// TIA Portal V21 export
FUNCTION "GestGruppoValvoleFestoVTEM" : Void   // FC68, LAD
{ S7_Optimized_Access := 'TRUE' }
// Ogni gruppo valvole festo può portare 8 valvole.
// Ognuno di qusti slot utilizza 3. word in lettura e 3 word in scrittura.
// 
// Se non vengono utilizzate 8 valvole è possibile sfruttura i moduli liberi per leggere dei dati dalle valvole. é anche possibile la lettura e scrittura ciclica delle informazioni.
// stored: SetENOAutomatically false
   VAR_INPUT
      HW_SUBMODULE : HW_SUBMODULE;
      SLOT01_K_Tipo : Int;
      SLOT01_K_UtenzaAttuatore : Int;   // Dichiarare la costante ad esempio k_valvolafestovftem oppure k_analogica da assegnare allo slot
      SLOT02_K_Tipo : Int;   // Dichiarare l'utilizzo dello slot, se deve essere utilizzato per leggere le informazioni dichiarare TipoAnalogica altrimenti valvola
      SLOT02_K_UtenzaAttuatore : Int;   // Dichiarare la costante ad esempio k_valvolafestovftem oppure k_analogica da assegnare allo slot
      SLOT03_K_Tipo : Int;   // Dichiarare l'utilizzo dello slot, se deve essere utilizzato per leggere le informazioni dichiarare TipoAnalogica altrimenti valvola
      SLOT03_K_UtenzaAttuatore : Int;   // Dichiarare la costante ad esempio k_valvolafestovftem oppure k_analogica da assegnare allo slot
      SLOT04_K_Tipo : Int;   // Dichiarare l'utilizzo dello slot, se deve essere utilizzato per leggere le informazioni dichiarare TipoAnalogica altrimenti valvola
      SLOT04_K_UtenzaAttuatore : Int;   // Dichiarare la costante ad esempio k_valvolafestovftem oppure k_analogica da assegnare allo slot
      SLOT05_K_Tipo : Int;   // Dichiarare l'utilizzo dello slot, se deve essere utilizzato per leggere le informazioni dichiarare TipoAnalogica altrimenti valvola
      SLOT05_K_UtenzaAttuatore : Int;   // Dichiarare la costante ad esempio k_valvolafestovftem oppure k_analogica da assegnare allo slot
      SLOT06_K_Tipo : Int;   // Dichiarare l'utilizzo dello slot, se deve essere utilizzato per leggere le informazioni dichiarare TipoAnalogica altrimenti valvola
      SLOT06_K_UtenzaAttuatore : Int;   // Dichiarare la costante ad esempio k_valvolafestovftem oppure k_analogica da assegnare allo slot
      SLOT07_K_Tipo : Int;   // Dichiarare l'utilizzo dello slot, se deve essere utilizzato per leggere le informazioni dichiarare TipoAnalogica altrimenti valvola
      SLOT07_K_UtenzaAttuatore : Int;   // Dichiarare la costante ad esempio k_valvolafestovftem oppure k_analogica da assegnare allo slot
      SLOT08_K_Tipo : Int;   // Dichiarare l'utilizzo dello slot, se deve essere utilizzato per leggere le informazioni dichiarare TipoAnalogica altrimenti valvola
      SLOT08_K_UtenzaAttuatore : Int;   // Dichiarare la costante ad esempio k_valvolafestovftem oppure k_analogica da assegnare allo slot
   END_VAR
   VAR_TEMP
      retval_1 : Int;
      retval_2 : Int;
      RispostaTelegramma : Array[0..23] of Word;
      InvioTelegramma : Array[0..23] of Word;
   END_VAR
BEGIN

REGION Network 1 (SCL): Gestione della comunicazione con ogni slot del gruppo.
   #retval_1 := DPRD_DAT(LADDR := #HW_SUBMODULE, RECORD => #RispostaTelegramma);

   "GestComunicazioneSlotVTEM"(K_UtenzaAttuatore:=#SLOT01_K_UtenzaAttuatore,
                               K_Tipo:=#SLOT01_K_Tipo,
                               NumeroSLOT:=1,
                               RispostaTelegramma:=#RispostaTelegramma,
                               InvioTelegramma=>#InvioTelegramma);
   "GestComunicazioneSlotVTEM"(K_UtenzaAttuatore := #SLOT02_K_UtenzaAttuatore,
                               K_Tipo := #SLOT02_K_Tipo,
                               NumeroSLOT := 2,
                               RispostaTelegramma := #RispostaTelegramma,
                               InvioTelegramma => #InvioTelegramma);
   "GestComunicazioneSlotVTEM"(K_UtenzaAttuatore := #SLOT03_K_UtenzaAttuatore,
                               K_Tipo := #SLOT03_K_Tipo,
                               NumeroSLOT := 3,
                               RispostaTelegramma := #RispostaTelegramma,
                               InvioTelegramma => #InvioTelegramma);
   "GestComunicazioneSlotVTEM"(K_UtenzaAttuatore := #SLOT04_K_UtenzaAttuatore,
                               K_Tipo := #SLOT04_K_Tipo,
                               NumeroSLOT := 4,
                               RispostaTelegramma := #RispostaTelegramma,
                               InvioTelegramma => #InvioTelegramma);
   "GestComunicazioneSlotVTEM"(K_UtenzaAttuatore := #SLOT05_K_UtenzaAttuatore,
                               K_Tipo := #SLOT05_K_Tipo,
                               NumeroSLOT := 5,
                               RispostaTelegramma := #RispostaTelegramma,
                               InvioTelegramma => #InvioTelegramma);
   "GestComunicazioneSlotVTEM"(K_UtenzaAttuatore := #SLOT06_K_UtenzaAttuatore,
                               K_Tipo := #SLOT06_K_Tipo,
                               NumeroSLOT := 6,
                               RispostaTelegramma := #RispostaTelegramma,
                               InvioTelegramma => #InvioTelegramma);
   "GestComunicazioneSlotVTEM"(K_UtenzaAttuatore := #SLOT07_K_UtenzaAttuatore,
                               K_Tipo := #SLOT07_K_Tipo,
                               NumeroSLOT := 7,
                               RispostaTelegramma := #RispostaTelegramma,
                               InvioTelegramma => #InvioTelegramma);
   "GestComunicazioneSlotVTEM"(K_UtenzaAttuatore := #SLOT08_K_UtenzaAttuatore,
                               K_Tipo := #SLOT08_K_Tipo,
                               NumeroSLOT := 8,
                               RispostaTelegramma := #RispostaTelegramma,
                               InvioTelegramma => #InvioTelegramma);

   #retval_2 := DPWR_DAT(LADDR := #HW_SUBMODULE, RECORD := #InvioTelegramma);
END_REGION
END_FUNCTION
